RoboDK station: ProgRob_stanica.rdk

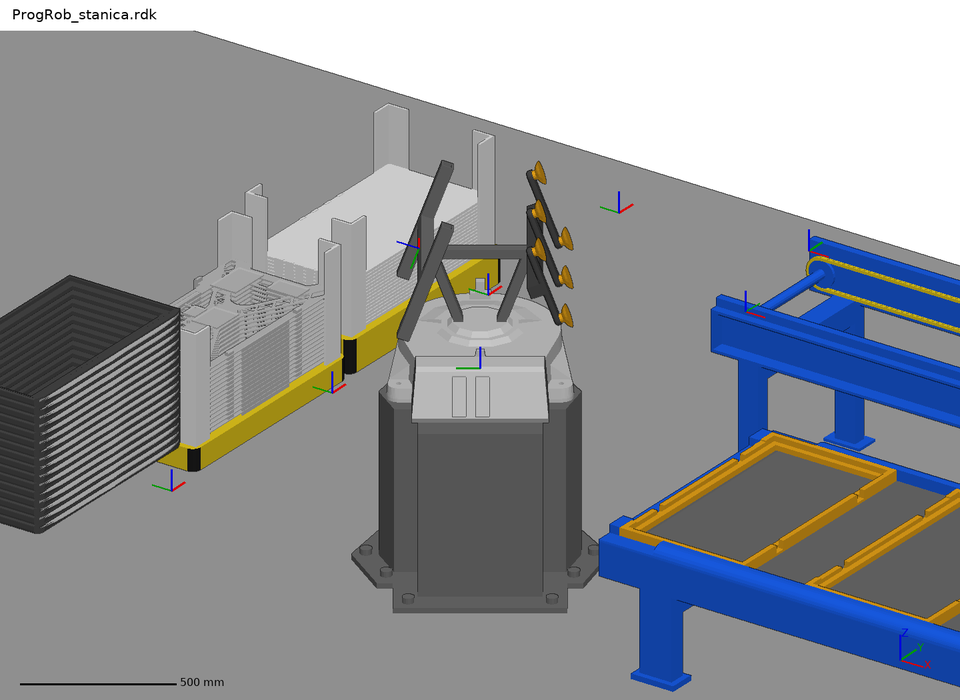
[picture v0: the station drawn from its stored meshes, robots at their saved joint values, targets as dots, program paths as lines]
Station ProgRob_stanica (saved by RoboDK 5.9.0). Poses are relative to the parent item; angles as X-Y-Z fixed-axis rotations.
Station parameters (name, value as stored): Assembly, 1, NextAssembly, 1, ScrewCircuit, 1, BuildCircuit, 1, UpFoamDone, 0, RackReady, 0, TAGS, ['Assembly']
  - frame TvRack_Rail at (-3000, 1420, 0) mm, rotated rx 0 ry 0 rz 90 deg
    - robot TvRack_Frame: 2 axes
        modified DH rows (alpha deg, a mm, theta deg, d mm): 0, 0, 0, 0 linear; 90, 0, 0, 0 linear
        base shift (0, 0, 0) mm, rotated rx 0 ry 90 rz 0 deg
        joint limits [-3250, -2100] to [0, 0]; home [0, 0]; saved at [-1600, 0]
      - frame TvRack_Frame_Ref at (0, 0, 0) mm
        - object TVFrame at (-750, 400, 0) mm, rotated rx 0 ry 0 rz -180 deg, size 786.6 x 406 x 28 mm, geometry from TVFrame.step
        - object TVFrame at (-750, 400, 15) mm, rotated rx 0 ry 0 rz -180 deg, size 786.6 x 406 x 28 mm, geometry from TVFrame.step
        - object TVFrame at (-750, 400, 30) mm, rotated rx 0 ry 0 rz -180 deg, size 786.6 x 406 x 28 mm, geometry from TVFrame.step
        - object TVFrame at (-750, 400, 45) mm, rotated rx 0 ry 0 rz -180 deg, size 786.6 x 406 x 28 mm, geometry from TVFrame.step
        - object TVFrame at (-750, 400, 60) mm, rotated rx 0 ry 0 rz -180 deg, size 786.6 x 406 x 28 mm, geometry from TVFrame.step
        - object TVFrame at (-750, 400, 75) mm, rotated rx 0 ry 0 rz -180 deg, size 786.6 x 406 x 28 mm, geometry from TVFrame.step
        - object TVFrame at (-750, 400, 90) mm, rotated rx 0 ry 0 rz -180 deg, size 786.6 x 406 x 28 mm, geometry from TVFrame.step
        - object TVFrame at (-750, 400, 105) mm, rotated rx 0 ry 0 rz -180 deg, size 786.6 x 406 x 28 mm, geometry from TVFrame.step
        - object TVFrame at (-750, 400, 120) mm, rotated rx 0 ry 0 rz -180 deg, size 786.6 x 406 x 28 mm, geometry from TVFrame.step
        - object TVFrame at (-750, 400, 135) mm, rotated rx 0 ry 0 rz -180 deg, size 786.6 x 406 x 28 mm, geometry from TVFrame.step
        - object TVFrame at (-750, 400, 225) mm, rotated rx 0 ry 0 rz -180 deg, size 786.6 x 406 x 28 mm, geometry from TVFrame.step
        - object TVFrame at (-750, 400, 210) mm, rotated rx 0 ry 0 rz -180 deg, size 786.6 x 406 x 28 mm, geometry from TVFrame.step
        - object TVFrame at (-750, 400, 195) mm, rotated rx 0 ry 0 rz -180 deg, size 786.6 x 406 x 28 mm, geometry from TVFrame.step
        - object TVFrame at (-750, 400, 180) mm, rotated rx 0 ry 0 rz -180 deg, size 786.6 x 406 x 28 mm, geometry from TVFrame.step
        - object TVFrame at (-750, 400, 165) mm, rotated rx 0 ry 0 rz -180 deg, size 786.6 x 406 x 28 mm, geometry from TVFrame.step
        - object TVFrame at (-750, 400, 150) mm, rotated rx 0 ry 0 rz -180 deg, size 786.6 x 406 x 28 mm, geometry from TVFrame.step
    - robot TvRack_Screen: 2 axes
        modified DH rows (alpha deg, a mm, theta deg, d mm): 0, 0, 0, 0 linear; 90, 0, 0, 0 linear
        base shift (0, 0, 0) mm, rotated rx 0 ry 90 rz 0 deg
        joint limits [-3250, -2100] to [0, 0]; home [0, 0]; saved at [-730, 0]
      - frame TvRack_Screen_Ref at (0, 0, 0) mm
        - object TVScreen at (0, 0, 0) mm, size 776.6 x 396 x 12 mm, geometry from TVScreen.step
        - object TVScreen at (0, 0, 12) mm, size 776.6 x 396 x 12 mm, geometry from TVScreen.step
        - object TVScreen at (0, 0, 24) mm, size 776.6 x 396 x 12 mm, geometry from TVScreen.step
        - object TVScreen at (0, 0, 36) mm, size 776.6 x 396 x 12 mm, geometry from TVScreen.step
        - object TVScreen at (0, 0, 48) mm, size 776.6 x 396 x 12 mm, geometry from TVScreen.step
        - object TVScreen at (0, 0, 60) mm, size 776.6 x 396 x 12 mm, geometry from TVScreen.step
        - object TVScreen at (0, 0, 72) mm, size 776.6 x 396 x 12 mm, geometry from TVScreen.step
        - object TVScreen at (0, 0, 84) mm, size 776.6 x 396 x 12 mm, geometry from TVScreen.step
        - object TVScreen at (0, 0, 96) mm, size 776.6 x 396 x 12 mm, geometry from TVScreen.step
        - object TVScreen at (0, 0, 108) mm, size 776.6 x 396 x 12 mm, geometry from TVScreen.step
        - object TVScreen at (0, 0, 120) mm, size 776.6 x 396 x 12 mm, geometry from TVScreen.step
        - object TVScreen at (0, 0, 132) mm, size 776.6 x 396 x 12 mm, geometry from TVScreen.step
        - object TVScreen at (0, 0, 144) mm, size 776.6 x 396 x 12 mm, geometry from TVScreen.step
        - object TVScreen at (0, 0, 180) mm, size 776.6 x 396 x 12 mm, geometry from TVScreen.step
        - object TVScreen at (0, 0, 168) mm, size 776.6 x 396 x 12 mm, geometry from TVScreen.step
        - object TVScreen at (0, 0, 156) mm, size 776.6 x 396 x 12 mm, geometry from TVScreen.step
    - frame TvRackFrontPanel Base at (-2480, 10, 0) mm
      - item type 7 TvRack_FrontPanel 1
      - item type 7 TvRack_FrontPanel 2
      - frame Frame 20 at (0, 0, 0) mm
        - object TVFrontPanel at (-750, 400, 0) mm, rotated rx 0 ry 0 rz 180 deg, size 812.6 x 460.3 x 32.5 mm, geometry from TVFrontCase.step
        - object TVFrontPanel at (-750, 400, 30) mm, rotated rx 0 ry 0 rz 180 deg, size 812.6 x 460.3 x 32.5 mm, geometry from TVFrontCase.step
        - object TVFrontPanel at (-750, 400, 60) mm, rotated rx 0 ry 0 rz 180 deg, size 812.6 x 460.3 x 32.5 mm, geometry from TVFrontCase.step
        - object TVFrontPanel at (-750, 400, 90) mm, rotated rx 0 ry 0 rz 180 deg, size 812.6 x 460.3 x 32.5 mm, geometry from TVFrontCase.step
        - object TVFrontPanel at (-750, 400, 120) mm, rotated rx 0 ry 0 rz 180 deg, size 812.6 x 460.3 x 32.5 mm, geometry from TVFrontCase.step
        - object TVFrontPanel at (-750, 400, 150) mm, rotated rx 0 ry 0 rz 180 deg, size 812.6 x 460.3 x 32.5 mm, geometry from TVFrontCase.step
        - object TVFrontPanel at (-750, 400, 180) mm, rotated rx 0 ry 0 rz 180 deg, size 812.6 x 460.3 x 32.5 mm, geometry from TVFrontCase.step
        - object TVFrontPanel at (-750, 400, 210) mm, rotated rx 0 ry 0 rz 180 deg, size 812.6 x 460.3 x 32.5 mm, geometry from TVFrontCase.step
        - object TVFrontPanel at (-750, 400, 270) mm, rotated rx 0 ry 0 rz 180 deg, size 812.6 x 460.3 x 32.5 mm, geometry from TVFrontCase.step
        - object TVFrontPanel at (-750, 400, 240) mm, rotated rx 0 ry 0 rz 180 deg, size 812.6 x 460.3 x 32.5 mm, geometry from TVFrontCase.step
        - object TVFrontPanel at (-750, 400, 300) mm, rotated rx 0 ry 0 rz 180 deg, size 812.6 x 460.3 x 32.5 mm, geometry from TVFrontCase.step
        - object TVFrontPanel at (-750, 400, 330) mm, rotated rx 0 ry 0 rz 180 deg, size 812.6 x 460.3 x 32.5 mm, geometry from TVFrontCase.step
        - object TVFrontPanel at (-750, 400, 360) mm, rotated rx 0 ry 0 rz 180 deg, size 812.6 x 460.3 x 32.5 mm, geometry from TVFrontCase.step
        - object TVFrontPanel at (-750, 400, 390) mm, rotated rx 0 ry 0 rz 180 deg, size 812.6 x 460.3 x 32.5 mm, geometry from TVFrontCase.step
        - object TVFrontPanel at (-750, 400, 420) mm, rotated rx 0 ry 0 rz 180 deg, size 812.6 x 460.3 x 32.5 mm, geometry from TVFrontCase.step
        - object TVFrontPanel at (-750, 400, 450) mm, rotated rx 0 ry 0 rz 180 deg, size 812.6 x 460.3 x 32.5 mm, geometry from TVFrontCase.step
  - frame MainConveyor Base at (-1580, 450, 650) mm
    - robot MainConveyor: 1 axes
        modified DH rows (alpha deg, a mm, theta deg, d mm): 0, 0, 0, 0 linear
        base shift (0, 0, 0) mm, rotated rx 0 ry 90 rz 0 deg
        joint limits [-200000] to [200000]; home [0]; saved at [0]
      - frame MainConveyorRef at (90, -480, 0) mm
        - object TVAssemblies at (2875, 462, 0) mm, rotated rx 0 ry 0 rz -180 deg, size 1893 x 485 x 64 mm
    - object Floor at (-100, -970, -650) mm, size 9000 x 4500 x 0 mm, geometry from Floor (2).sld
  - frame ABB IRB 2400/16 Base at (-2010, -770, 600) mm, rotated rx 0 ry 0 rz 125 deg
    - robot ABB IRB 2400/16: 6 axes, payload 16 kg, reach 1550 mm, repeatability 0.03 mm, weight 380 kg
        joint limits [-180, -100, -60, -200, -120, -400] to [180, 110, 65, 200, 120, 400]; home [0, 0, 0, 0, 0, 0]; saved at [-92.609, 38.532, 58.57, -72.434, -56.335, -58.059]
      - frame ToolRobot1 Base at (0, 195, 425) mm, rotated rx -70 ry 0 rz 0 deg
        - robot ToolRobot1: 1 axes
            joint limits [-20] to [200]; home [0]; saved at [26]
      - tool ToolRobot1_TCP_Gripper, TCP at (0, 195, 425) mm, rotated rx -70 ry 0 rz 0 deg
      - tool ToolRobot1_TCP_Cup, TCP at (0, -240, 450) mm, rotated rx 70 ry 0 rz 0 deg
    - object Robot1_Stand at (0, 0, 0) mm, size 938.8 x 824.6 x 600 mm, geometry from Robot1_Stand.step
  - frame AssemblyRackConveyor Base at (1530, -1260, 440) mm
    - robot AssemblyRackConveyor: 1 axes
        modified DH rows (alpha deg, a mm, theta deg, d mm): 0, 0, 0, 0 linear
        base shift (0, 0, 0) mm, rotated rx 0 ry 90 rz 0 deg
        joint limits [-200000] to [200000]; home [0]; saved at [0]
      - frame AssemblyRackConveyorRef at (0, 0, 0) mm
        - object AssemblyRack at (-1440, 0, 0) mm, size 40 x 853 x 485 mm, geometry from AssemblyRack.step
        - object AssemblyRack at (-720, 0, 0) mm, size 40 x 853 x 485 mm, geometry from AssemblyRack.step
        - object AssemblyRack at (-2160, 0, 0) mm, size 40 x 853 x 485 mm, geometry from AssemblyRack.step
